(*
    Function block for a single Solid ATTenuator (SATT) filter stack
    under the LCLS_Tc_Motion (ND) framework. This is for the L2SI
    compact design with 4 filter stacks that each have many filters.

    Single-axis Y mover with nine states (OUT, FILTER1..FILTER8) via
    FB_PositionStateND. SATT is **not** a PMPS state mover: there is
    no arbiter handshake, no BPTM, no beam-param gating, no
    transition-key plumbing, no eMotionRequestPolicy other than the
    default. The only PMPS-adjacent behavior is:
      - Reactive temperature setpoint pulled from the PMPS JSON DB by
        an in-device FB_JsonDocToSafeBP read keyed on the caller-
        supplied RTDPMPSState, used as the two RTD fault thresholds.
      - A single FB_FastFault ("Device is moving") raised whenever
        the stage is in motion or in UNKNOWN, sunk into the caller-
        supplied fbFFHWO.

    Transmission for the stack's currently selected filter is
    calculated each cycle from arrFilters[iFilterIndex] (material,
    thickness), the current beam energy
    (PMPS_GVL.stCurrentBeamParameters.neV), and the per-element
    atomic-mass + density lookups (FB_AtomicMass /
    FB_AttenuatorElementDensity).

    Caller responsibilities:
      - Own and tick FB_MotionStageNC for the Y motor; pass it into
        aiMotionStage via FB_Init.
      - Own astPositionState[1..MAX_STATE_MOTORS][1..MAX_STATES] and
        configure each state's sName + fPosition (+ fDelta) in the
        caller app before calling fbSATT (only stack-slot 1 matters
        for SATT). The filters are not real PMPS states, so the
        per-filter stPMPS.sPmpsState is not used.
      - Own fbFFHWO (caller-side hardware fast-fault sink).
      - Set sDeviceName (used for both DB lookup and FF messages) and
        RTDPMPSState (the PMPS DB key for the RTD reactive-temperature
        read), both passed via FB_Init.
*)
{attribute 'call_after_init'}
FUNCTION_BLOCK FB_SXR_SATT_Stage
VAR_INPUT
    (* Device-specific state-enum bridges. Typed as
       E_SXR_SATT_Position (UINT base) so the caller surface is enum-
       checked; the inline-init below binds them to
       FB_PositionStateND's REFERENCE TO UINT params via the shared
       UINT base. Callers drive moves with
       `fbSATT.eEnumSet := E_SXR_SATT_Position.FILTER1;`. *)
    eEnumSet : E_SXR_SATT_Position;
    eEnumGet : E_SXR_SATT_Position;

    (* Per-filter material / thickness table. Used by the transmission
       calculation. Index 1 corresponds to FILTER1 (which is the
       state at slot 2 in astPositionState, since OUT lives at slot 1
       in E_SXR_SATT_Position). *)
    {attribute 'pytmc' := 'pv: FILTERS'}
    arrFilters : ARRAY[1..8] OF ST_SATT_Filter;
END_VAR
VAR_OUTPUT
    fTemp1                    : LREAL;
    fTemp2                    : LREAL;
    bIsStationary             : BOOL;
    bError                    : BOOL;

    {attribute 'pytmc' := '
        pv: MATERIAL
        io: i
    '}
    sActiveFilterMaterial     : STRING;

    {attribute 'pytmc' := '
        pv: THICKNESS
        io: i
        field: EGU um
    '}
    fActiveFilterThickness_um : LREAL;

    {attribute 'pytmc' := '
        pv: TRANSMISSION
        io: i
        field: DESC Filter transmission
    '}
    fTransmission             : LREAL;
    fActiveFilterDensity      : LREAL;
    fActiveFilterAtomicMass   : LREAL;
    fAbsorptionConstant       : LREAL;

    iFilterIndex              : INT := 0;
END_VAR
VAR
    fbStates : FB_PositionStateND(
        aiMotionStage        := aiMotionStage,
        astPositionState     := astPositionState,
        nActiveMotorCount    := 1,
        eEnumSet             := eEnumSet,
        eEnumGet             := eEnumGet,
        bEnableMotion        := bEnableMotion,
        eMotionRequestPolicy := E_MotionRequestPolicy.INTERRUPT
    );

    fbAtomicMass               : FB_AtomicMass;
    fbAttenuatorElementDensity : FB_AttenuatorElementDensity;

    (* EL3202-0020: 0.01 deg C per digit. Vetoed when the stage is in
       OUT (no filter in beam, no temperature to monitor). *)
    {attribute 'pytmc' := 'pv: RTD:1'}
    fbRTD_1 : FB_CC_TempSensor := (fResolution := 0.01);
    {attribute 'pytmc' := 'pv: RTD:2'}
    fbRTD_2 : FB_CC_TempSensor := (fResolution := 0.01);

    bFileReaderBusy       : REFERENCE TO BOOL;
    (* Per-cycle JSON DB read for the currently active filter's
       PMPS state, just to pull the reactive temp setpoint into
       astPickedDB[1].stReactiveParams.nTempSP. Not a PMPS BPTM
       participant; just borrows the DB pipeline. *)
    fbReadPMPSDB : FB_JsonDocToSafeBP;
    astPickedDB  : ARRAY[1..1] OF ST_DbStateParams;

    (* "Device is moving" fast fault. Raised while the Y motor is
       moving or while we are sitting in UNKNOWN. *)
    fbFF : FB_FastFault := (
        i_Desc       := 'Device is moving',
        i_TypeCode   := E_MotionFFType.DEVICE_MOVE,
        i_xAutoReset := TRUE
    );

    (* REFERENCE TO backing fields populated by FB_Init. Same names as
       FB_Init params; THIS^. disambiguates inside FB_Init.
       Live-bound to caller storage for the lifetime of the FB. *)
    {attribute 'no_copy'}
    aiMotionStage    : REFERENCE TO ARRAY[1..MotionConstants.MAX_STATE_MOTORS] OF I_MotionStage;
    {attribute 'no_copy'}
    astPositionState : REFERENCE TO ARRAY[1..MotionConstants.MAX_STATE_MOTORS]
                                          OF ARRAY[1..GeneralConstants.MAX_STATES] OF ST_PositionState;
    {attribute 'no_copy'}
    fbFFHWO          : REFERENCE TO FB_HardwareFFOutput;
    sDeviceName      : STRING;
    (* PMPS DB key for the RTD reactive-temperature read. The filters
       are not real PMPS states, so this device-level key (caller-
       supplied via FB_Init) names the DB entry to pull the reactive
       temp setpoint from. *)
    RTDPMPSState     : STRING;
    bEnableMotion    : BOOL := TRUE;
END_VAR

(* Nil-ref guards: every REFERENCE TO backing field must be bound. *)
IF NOT __ISVALIDREF(aiMotionStage)
   OR NOT __ISVALIDREF(astPositionState)
   OR NOT __ISVALIDREF(fbFFHWO) THEN
    RETURN;
END_IF

fbStates();

(* Filter index is offset by one because E_SXR_SATT_Position.OUT
   occupies slot 1 and FILTER1..FILTER8 occupy slots 2..9. *)
iFilterIndex := UINT_TO_INT(eEnumGet) - 1;

IF iFilterIndex >= 1 AND iFilterIndex <= 8 THEN
    sActiveFilterMaterial     := arrFilters[iFilterIndex].sFilterMaterial;
    fActiveFilterThickness_um := arrFilters[iFilterIndex].fFilterThickness_um;

    fbAtomicMass(
        sName  := sActiveFilterMaterial,
        fValue => fActiveFilterAtomicMass
    );
    fbAttenuatorElementDensity(
        sName    := sActiveFilterMaterial,
        fDensity => fActiveFilterDensity
    );

    fAbsorptionConstant := F_CalculateAbsorptionConstant(
        sElement      := sActiveFilterMaterial,
        fEnergyEV     := PMPS_GVL.stCurrentBeamParameters.neV,
        fDensity_gm3  := fActiveFilterDensity,
        fAtomicWeight := fActiveFilterAtomicMass,
        bError        => bError
    );
    fTransmission := F_CalculateTransmission(
        fAbsorptionConstant := fAbsorptionConstant,
        fThickness_in_m     := fActiveFilterThickness_um * 1.0E-6
    );
ELSE
    sActiveFilterMaterial     := '';
    fActiveFilterThickness_um := 0.0;
    fAbsorptionConstant       := 0.0;
    fActiveFilterDensity      := 0.0;
    fActiveFilterAtomicMass   := 0.0;
    fTransmission             := 1.0;
END_IF

(* "Device is moving" fault: stationary AND known position. Reads the
   motor's NC status through the I_MotionStage interface; aiMotionStage
   was nil-guarded above so slot 1 deref is safe. *)
bIsStationary := NOT aiMotionStage[1].Axis.Status.Moving;
fbFF(
    i_DevName  := sDeviceName,
    i_xOK      := bIsStationary AND eEnumGet <> E_SXR_SATT_Position.UNKNOWN,
    io_fbFFHWO := fbFFHWO
);

(* The RTD reactive-temperature read is keyed on the device-level
   RTDPMPSState (the filters are not real PMPS states, so no per-
   filter key is scanned). The named DB entry must exist; the
   temperature field may be blank. *)
astPickedDB[1].sPmpsState := RTDPMPSState;

fbReadPMPSDB(
    bExecute    := NOT bFileReaderBusy,
    jsonDoc     := PMPS_GVL.BP_jsonDoc,
    sDeviceName := sDeviceName,
    arrStates   := astPickedDB,
    io_fbFFHWO  := fbFFHWO
);

fbRTD_1(
    fFaultThreshold := astPickedDB[1].stReactiveParams.nTempSP,
    sDevName        := sDeviceName,
    bVeto           := eEnumGet = E_SXR_SATT_Position.OUT,
    io_fbFFHWO      := fbFFHWO
);
fTemp1 := fbRTD_1.fTemp;

fbRTD_2(
    fFaultThreshold := astPickedDB[1].stReactiveParams.nTempSP,
    sDevName        := sDeviceName,
    bVeto           := eEnumGet = E_SXR_SATT_Position.OUT,
    io_fbFFHWO      := fbFFHWO
);
fTemp2 := fbRTD_2.fTemp;

(*
    {attribute 'call_after_init'} on FB_SXR_SATT_Stage causes TwinCAT
    to auto-fire THIS^.CallAfterInit() after FB_SXR_SATT_Stage.FB_Init
    completes.

    fbStates was constructed via inline-init in this FB's VAR section,
    which ran BEFORE FB_Init bound the REF fields on THIS^.
    Consequently fbStates' inline-init forwarded nil REFs into
    fbStates.FB_Init, and the auto-fired fbStates.CallAfterInit guards
    on those nil REFs and bails. This method re-supplies the now-valid
    refs through fbStates.CallAfterInitStateMover, which re-binds them and
    runs the Core / ND child-FB wiring chain.
*)
{attribute 'call_after_init'}
METHOD CallAfterInit
THIS^.fbStates.CallAfterInitStateMover(
    aiMotionStage         := aiMotionStage,
    astPositionState      := astPositionState,
    nActiveMotorCount     := 1,
    eEnumSet              := eEnumSet,
    eEnumGet              := eEnumGet,
    bEnableMotion         := bEnableMotion,
    eMotionRequestPolicy  := E_MotionRequestPolicy.INTERRUPT,
);
END_METHOD

(* Stores all FB_Init inputs into instance fields. Every input is
   REFERENCE TO and is REF= bound for the lifetime of the FB.
   Inline-init of fbStates above runs first, capturing the FB_Init
   params at construction time; this method then records the same
   references on THIS^ for body-side use and live caller writes. *)
{attribute 'analysis' := '-33'}
METHOD FB_Init : BOOL
VAR_INPUT
    bInitRetains     : BOOL;
    bInCopyCode      : BOOL;
    aiMotionStage    : REFERENCE TO ARRAY[1..MotionConstants.MAX_STATE_MOTORS] OF I_MotionStage;
    astPositionState : REFERENCE TO ARRAY[1..MotionConstants.MAX_STATE_MOTORS]
                                          OF ARRAY[1..GeneralConstants.MAX_STATES] OF ST_PositionState;
    bFileReaderBusy       : REFERENCE TO BOOL;
    fbFFHWO          : REFERENCE TO FB_HardwareFFOutput;
    sDeviceName      : STRING;
    RTDPMPSState     : STRING;
END_VAR
THIS^.aiMotionStage    REF= aiMotionStage;
THIS^.astPositionState REF= astPositionState;
THIS^.fbFFHWO          REF= fbFFHWO;
THIS^.bFileReaderBusy 	REF=bFileReaderBusy;
THIS^.sDeviceName      := sDeviceName;
THIS^.RTDPMPSState     := RTDPMPSState;
END_METHOD

END_FUNCTION_BLOCK

(* stored: Version 1.1.0.1
   POU FB_SXR_SATT_Stage: Id {7fb611c7-2215-4e8f-8a28-e51a98acae9a}, SpecialFunc None
   Method CallAfterInit: Id {7fb611c8-2215-4e8f-8a28-e51a98acae9b}
   Method FB_init: Id {7fb611c9-2215-4e8f-8a28-e51a98acae9c} *)
